// Mitsubishi GX Works2 project: Project-2_찐   PLC: Q03UD

PROGRAM AGV
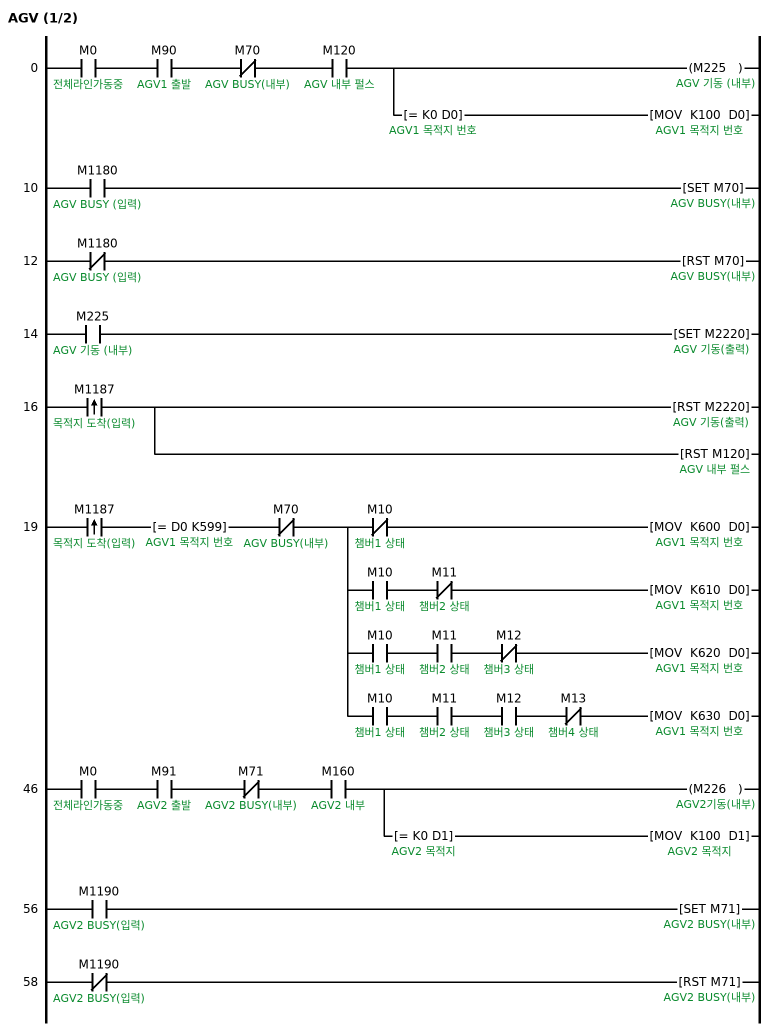
0     LD      M0  ; 전체라인가동중
      AND     M90  ; AGV1 출발
      ANI     M70  ; AGV BUSY(내부)
      AND     M120  ; AGV 내부 펄스
      OUT     M225  ; AGV 기동 (내부)
      AND=    K0 D0  ; AGV1 목적지 번호
      MOV     K100 D0
10    LD      M1180  ; AGV BUSY (입력)
      SET     M70  ; AGV BUSY(내부)
12    LDI     M1180  ; AGV BUSY (입력)
      RST     M70  ; AGV BUSY(내부)
14    LD      M225  ; AGV 기동 (내부)
      SET     M2220  ; AGV 기동(출력)
16    LDP     M1187  ; 목적지 도착(입력)
      RST     M2220  ; AGV 기동(출력)
      RST     M120  ; AGV 내부 펄스
19    LDP     M1187  ; 목적지 도착(입력)
      AND=    D0 K599  ; AGV1 목적지 번호
      ANI     M70  ; AGV BUSY(내부)
      MPS
      ANI     M10  ; 챔버1 상태
      MOV     K600 D0
      MRD
      AND     M10  ; 챔버1 상태
      ANI     M11  ; 챔버2 상태
      MOV     K610 D0
      MRD
      AND     M10  ; 챔버1 상태
      AND     M11  ; 챔버2 상태
      ANI     M12  ; 챔버3 상태
      MOV     K620 D0
      MPP
      AND     M10  ; 챔버1 상태
      AND     M11  ; 챔버2 상태
      AND     M12  ; 챔버3 상태
      ANI     M13  ; 챔버4 상태
      MOV     K630 D0
46    LD      M0  ; 전체라인가동중
      AND     M91  ; AGV2 출발
      ANI     M71  ; AGV2 BUSY(내부)
      AND     M160  ; AGV2 내부
      OUT     M226  ; AGV2기동(내부)
      AND=    K0 D1  ; AGV2 목적지
      MOV     K100 D1
56    LD      M1190  ; AGV2 BUSY(입력)
      SET     M71  ; AGV2 BUSY(내부)
58    LDI     M1190  ; AGV2 BUSY(입력)
      RST     M71  ; AGV2 BUSY(내부)
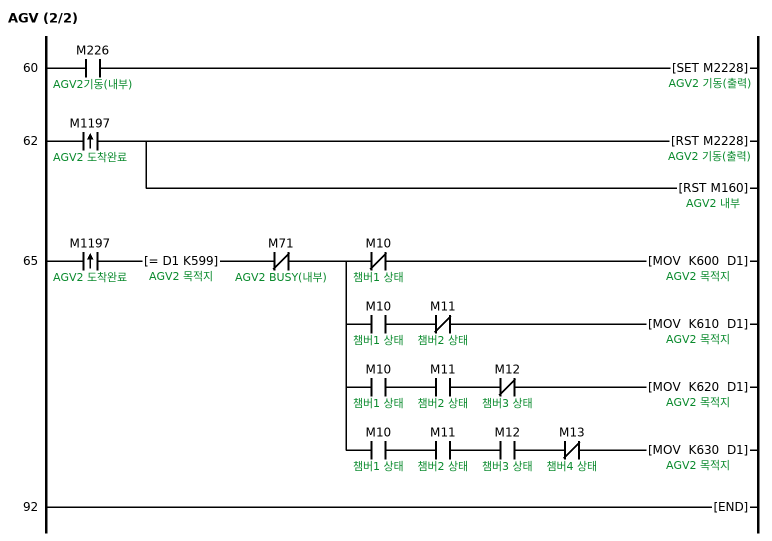
60    LD      M226  ; AGV2기동(내부)
      SET     M2228  ; AGV2 기동(출력)
62    LDP     M1197  ; AGV2 도착완료
      RST     M2228  ; AGV2 기동(출력)
      RST     M160  ; AGV2 내부
65    LDP     M1197  ; AGV2 도착완료
      AND=    D1 K599  ; AGV2 목적지
      ANI     M71  ; AGV2 BUSY(내부)
      MPS
      ANI     M10  ; 챔버1 상태
      MOV     K600 D1
      MRD
      AND     M10  ; 챔버1 상태
      ANI     M11  ; 챔버2 상태
      MOV     K610 D1
      MRD
      AND     M10  ; 챔버1 상태
      AND     M11  ; 챔버2 상태
      ANI     M12  ; 챔버3 상태
      MOV     K620 D1
      MPP
      AND     M10  ; 챔버1 상태
      AND     M11  ; 챔버2 상태
      AND     M12  ; 챔버3 상태
      ANI     M13  ; 챔버4 상태
      MOV     K630 D1
92    END
END_PROGRAM

PROGRAM Check_4
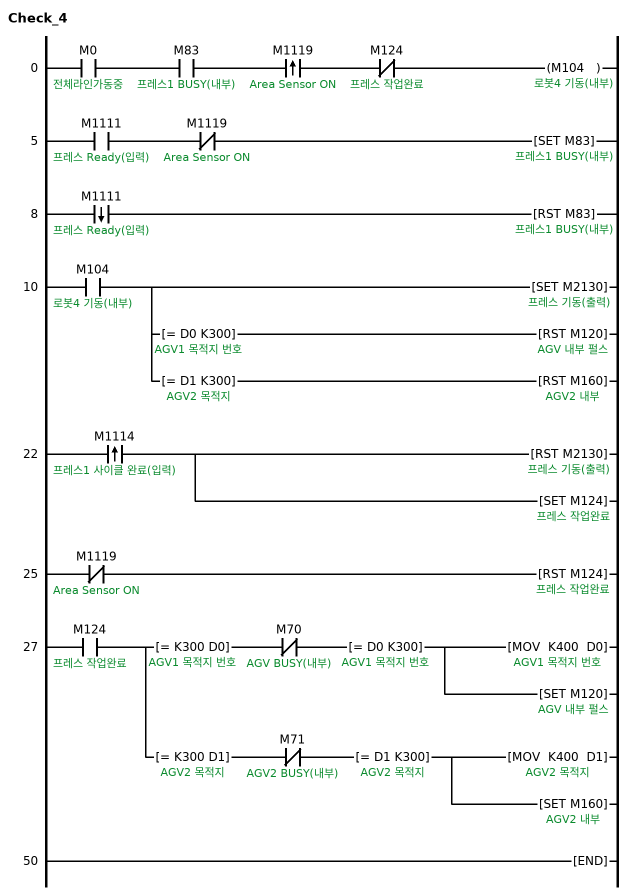
0     LD      M0  ; 전체라인가동중
      AND     M83  ; 프레스1 BUSY(내부)
      ANDP    M1119  ; Area Sensor ON
      ANI     M124  ; 프레스 작업완료
      OUT     M104  ; 로봇4 기동(내부)
5     LD      M1111  ; 프레스 Ready(입력)
      ANI     M1119  ; Area Sensor ON
      SET     M83  ; 프레스1 BUSY(내부)
8     LDF     M1111  ; 프레스 Ready(입력)
      RST     M83  ; 프레스1 BUSY(내부)
10    LD      M104  ; 로봇4 기동(내부)
      SET     M2130  ; 프레스 기동(출력)
      MPS
      AND=    D0 K300  ; AGV1 목적지 번호
      RST     M120  ; AGV 내부 펄스
      MPP
      AND=    D1 K300  ; AGV2 목적지
      RST     M160  ; AGV2 내부
22    LDP     M1114  ; 프레스1 사이클 완료(입력)
      RST     M2130  ; 프레스 기동(출력)
      SET     M124  ; 프레스 작업완료
25    LDI     M1119  ; Area Sensor ON
      RST     M124  ; 프레스 작업완료
27    LD      M124  ; 프레스 작업완료
      MPS
      AND=    K300 D0  ; AGV1 목적지 번호
      ANI     M70  ; AGV BUSY(내부)
      AND=    D0 K300  ; AGV1 목적지 번호
      MOV     K400 D0
      SET     M120  ; AGV 내부 펄스
      MPP
      AND=    K300 D1  ; AGV2 목적지
      ANI     M71  ; AGV2 BUSY(내부)
      AND=    D1 K300  ; AGV2 목적지
      MOV     K400 D1
      SET     M160  ; AGV2 내부
50    END
END_PROGRAM

PROGRAM MAIN
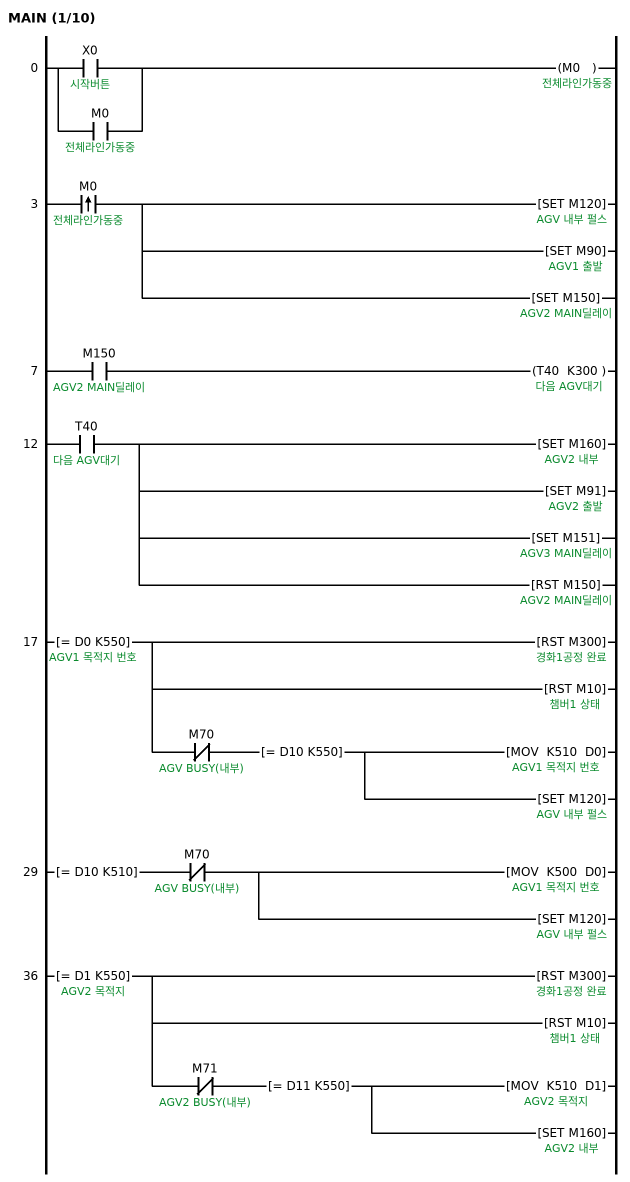
0     LD      X0  ; 시작버튼
      OR      M0  ; 전체라인가동중
      OUT     M0  ; 전체라인가동중
3     LDP     M0  ; 전체라인가동중
      SET     M120  ; AGV 내부 펄스
      SET     M90  ; AGV1 출발
      SET     M150  ; AGV2 MAIN딜레이
7     LD      M150  ; AGV2 MAIN딜레이
      OUT     T40 K300  ; 다음 AGV대기
12    LD      T40  ; 다음 AGV대기
      SET     M160  ; AGV2 내부
      SET     M91  ; AGV2 출발
      SET     M151  ; AGV3 MAIN딜레이
      RST     M150  ; AGV2 MAIN딜레이
17    LD=     D0 K550  ; AGV1 목적지 번호
      RST     M300  ; 경화1공정 완료
      RST     M10  ; 챔버1 상태
      ANI     M70  ; AGV BUSY(내부)
      AND=    D10 K550
      MOV     K510 D0
      SET     M120  ; AGV 내부 펄스
29    LD=     D10 K510
      ANI     M70  ; AGV BUSY(내부)
      MOV     K500 D0
      SET     M120  ; AGV 내부 펄스
36    LD=     D1 K550  ; AGV2 목적지
      RST     M300  ; 경화1공정 완료
      RST     M10  ; 챔버1 상태
      ANI     M71  ; AGV2 BUSY(내부)
      AND=    D11 K550
      MOV     K510 D1
      SET     M160  ; AGV2 내부
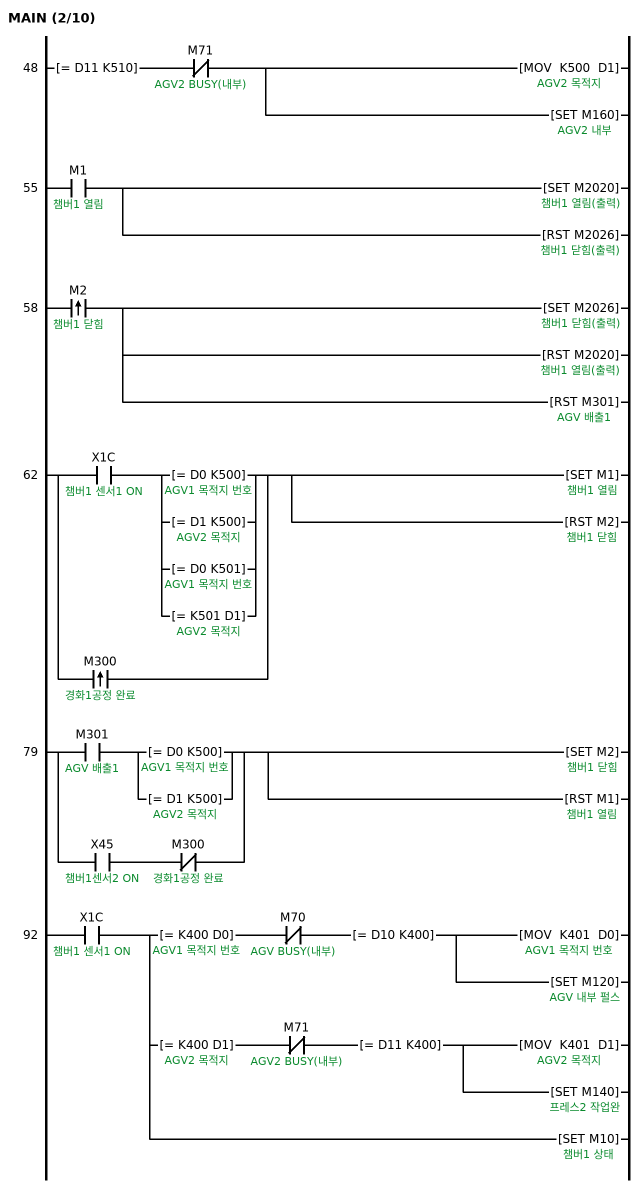
48    LD=     D11 K510
      ANI     M71  ; AGV2 BUSY(내부)
      MOV     K500 D1
      SET     M160  ; AGV2 내부
55    LD      M1  ; 챔버1 열림
      SET     M2020  ; 챔버1 열림(출력)
      RST     M2026  ; 챔버1 닫힘(출력)
58    LDP     M2  ; 챔버1 닫힘
      SET     M2026  ; 챔버1 닫힘(출력)
      RST     M2020  ; 챔버1 열림(출력)
      RST     M301  ; AGV 배출1
62    LD      X1C  ; 챔버1 센서1 ON
      LD=     D0 K500  ; AGV1 목적지 번호
      OR=     D1 K500  ; AGV2 목적지
      OR=     D0 K501  ; AGV1 목적지 번호
      OR=     K501 D1  ; AGV2 목적지
      ANB
      ORP     M300  ; 경화1공정 완료
      SET     M1  ; 챔버1 열림
      RST     M2  ; 챔버1 닫힘
79    LD      M301  ; AGV 배출1
      LD=     D0 K500  ; AGV1 목적지 번호
      OR=     D1 K500  ; AGV2 목적지
      ANB
      LD      X45  ; 챔버1센서2 ON
      ANI     M300  ; 경화1공정 완료
      ORB
      SET     M2  ; 챔버1 닫힘
      RST     M1  ; 챔버1 열림
92    LD      X1C  ; 챔버1 센서1 ON
      MPS
      AND=    K400 D0  ; AGV1 목적지 번호
      ANI     M70  ; AGV BUSY(내부)
      AND=    D10 K400
      MOV     K401 D0
      SET     M120  ; AGV 내부 펄스
      MRD
      AND=    K400 D1  ; AGV2 목적지
      ANI     M71  ; AGV2 BUSY(내부)
      AND=    D11 K400
      MOV     K401 D1
      SET     M140  ; 프레스2 작업완
      MPP
      SET     M10  ; 챔버1 상태
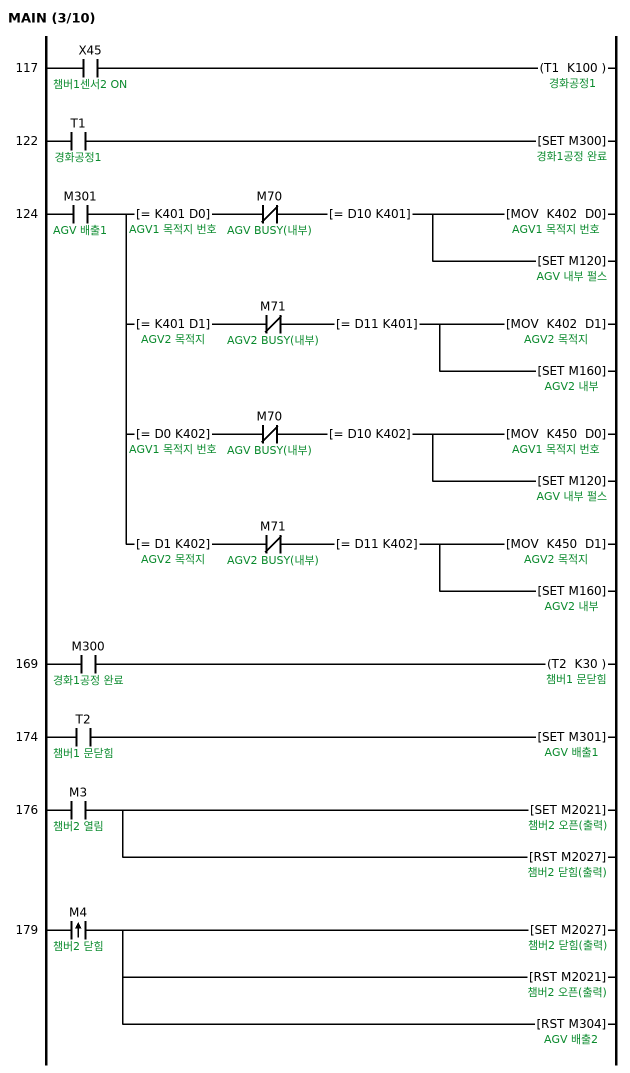
117   LD      X45  ; 챔버1센서2 ON
      OUT     T1 K100  ; 경화공정1
122   LD      T1  ; 경화공정1
      SET     M300  ; 경화1공정 완료
124   LD      M301  ; AGV 배출1
      MPS
      AND=    K401 D0  ; AGV1 목적지 번호
      ANI     M70  ; AGV BUSY(내부)
      AND=    D10 K401
      MOV     K402 D0
      SET     M120  ; AGV 내부 펄스
      MRD
      AND=    K401 D1  ; AGV2 목적지
      ANI     M71  ; AGV2 BUSY(내부)
      AND=    D11 K401
      MOV     K402 D1
      SET     M160  ; AGV2 내부
      MRD
      AND=    D0 K402  ; AGV1 목적지 번호
      ANI     M70  ; AGV BUSY(내부)
      AND=    D10 K402
      MOV     K450 D0
      SET     M120  ; AGV 내부 펄스
      MPP
      AND=    D1 K402  ; AGV2 목적지
      ANI     M71  ; AGV2 BUSY(내부)
      AND=    D11 K402
      MOV     K450 D1
      SET     M160  ; AGV2 내부
169   LD      M300  ; 경화1공정 완료
      OUT     T2 K30  ; 챔버1 문닫힘
174   LD      T2  ; 챔버1 문닫힘
      SET     M301  ; AGV 배출1
176   LD      M3  ; 챔버2 열림
      SET     M2021  ; 챔버2 오픈(출력)
      RST     M2027  ; 챔버2 닫힘(출력)
179   LDP     M4  ; 챔버2 닫힘
      SET     M2027  ; 챔버2 닫힘(출력)
      RST     M2021  ; 챔버2 오픈(출력)
      RST     M304  ; AGV 배출2
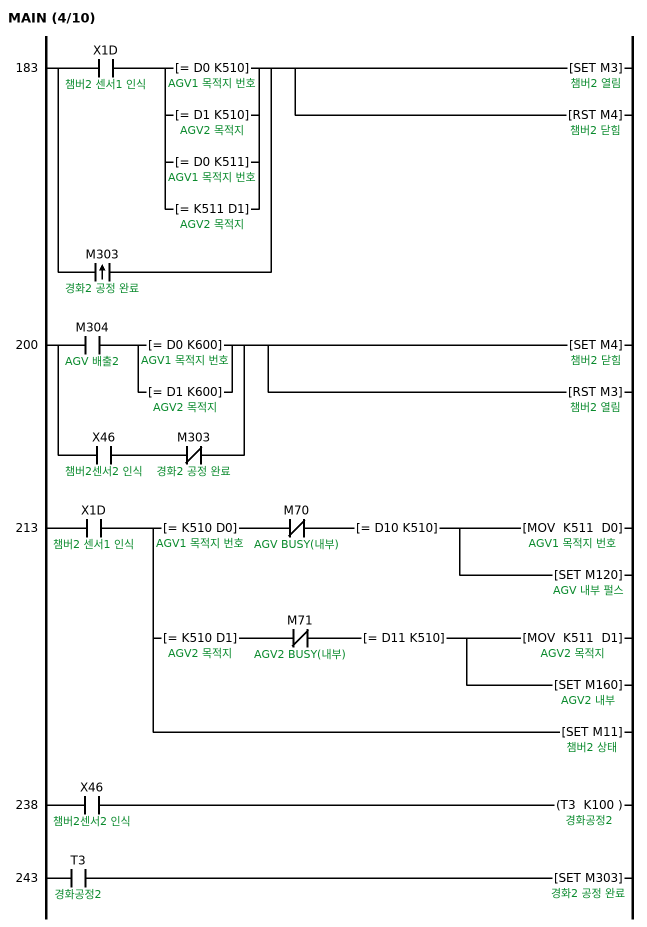
183   LD      X1D  ; 챔버2 센서1 인식
      LD=     D0 K510  ; AGV1 목적지 번호
      OR=     D1 K510  ; AGV2 목적지
      OR=     D0 K511  ; AGV1 목적지 번호
      OR=     K511 D1  ; AGV2 목적지
      ANB
      ORP     M303  ; 경화2 공정 완료
      SET     M3  ; 챔버2 열림
      RST     M4  ; 챔버2 닫힘
200   LD      M304  ; AGV 배출2
      LD=     D0 K600  ; AGV1 목적지 번호
      OR=     D1 K600  ; AGV2 목적지
      ANB
      LD      X46  ; 챔버2센서2 인식
      ANI     M303  ; 경화2 공정 완료
      ORB
      SET     M4  ; 챔버2 닫힘
      RST     M3  ; 챔버2 열림
213   LD      X1D  ; 챔버2 센서1 인식
      MPS
      AND=    K510 D0  ; AGV1 목적지 번호
      ANI     M70  ; AGV BUSY(내부)
      AND=    D10 K510
      MOV     K511 D0
      SET     M120  ; AGV 내부 펄스
      MRD
      AND=    K510 D1  ; AGV2 목적지
      ANI     M71  ; AGV2 BUSY(내부)
      AND=    D11 K510
      MOV     K511 D1
      SET     M160  ; AGV2 내부
      MPP
      SET     M11  ; 챔버2 상태
238   LD      X46  ; 챔버2센서2 인식
      OUT     T3 K100  ; 경화공정2
243   LD      T3  ; 경화공정2
      SET     M303  ; 경화2 공정 완료
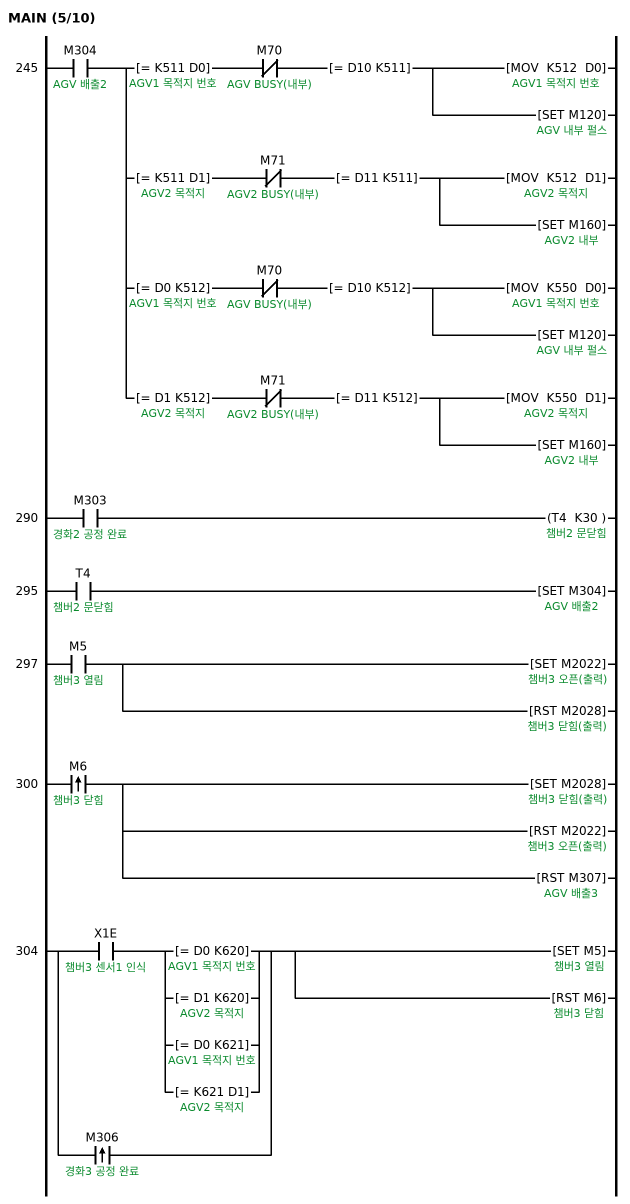
245   LD      M304  ; AGV 배출2
      MPS
      AND=    K511 D0  ; AGV1 목적지 번호
      ANI     M70  ; AGV BUSY(내부)
      AND=    D10 K511
      MOV     K512 D0
      SET     M120  ; AGV 내부 펄스
      MRD
      AND=    K511 D1  ; AGV2 목적지
      ANI     M71  ; AGV2 BUSY(내부)
      AND=    D11 K511
      MOV     K512 D1
      SET     M160  ; AGV2 내부
      MRD
      AND=    D0 K512  ; AGV1 목적지 번호
      ANI     M70  ; AGV BUSY(내부)
      AND=    D10 K512
      MOV     K550 D0
      SET     M120  ; AGV 내부 펄스
      MPP
      AND=    D1 K512  ; AGV2 목적지
      ANI     M71  ; AGV2 BUSY(내부)
      AND=    D11 K512
      MOV     K550 D1
      SET     M160  ; AGV2 내부
290   LD      M303  ; 경화2 공정 완료
      OUT     T4 K30  ; 챔버2 문닫힘
295   LD      T4  ; 챔버2 문닫힘
      SET     M304  ; AGV 배출2
297   LD      M5  ; 챔버3 열림
      SET     M2022  ; 챔버3 오픈(출력)
      RST     M2028  ; 챔버3 닫힘(출력)
300   LDP     M6  ; 챔버3 닫힘
      SET     M2028  ; 챔버3 닫힘(출력)
      RST     M2022  ; 챔버3 오픈(출력)
      RST     M307  ; AGV 배출3
304   LD      X1E  ; 챔버3 센서1 인식
      LD=     D0 K620  ; AGV1 목적지 번호
      OR=     D1 K620  ; AGV2 목적지
      OR=     D0 K621  ; AGV1 목적지 번호
      OR=     K621 D1  ; AGV2 목적지
      ANB
      ORP     M306  ; 경화3 공정 완료
      SET     M5  ; 챔버3 열림
      RST     M6  ; 챔버3 닫힘
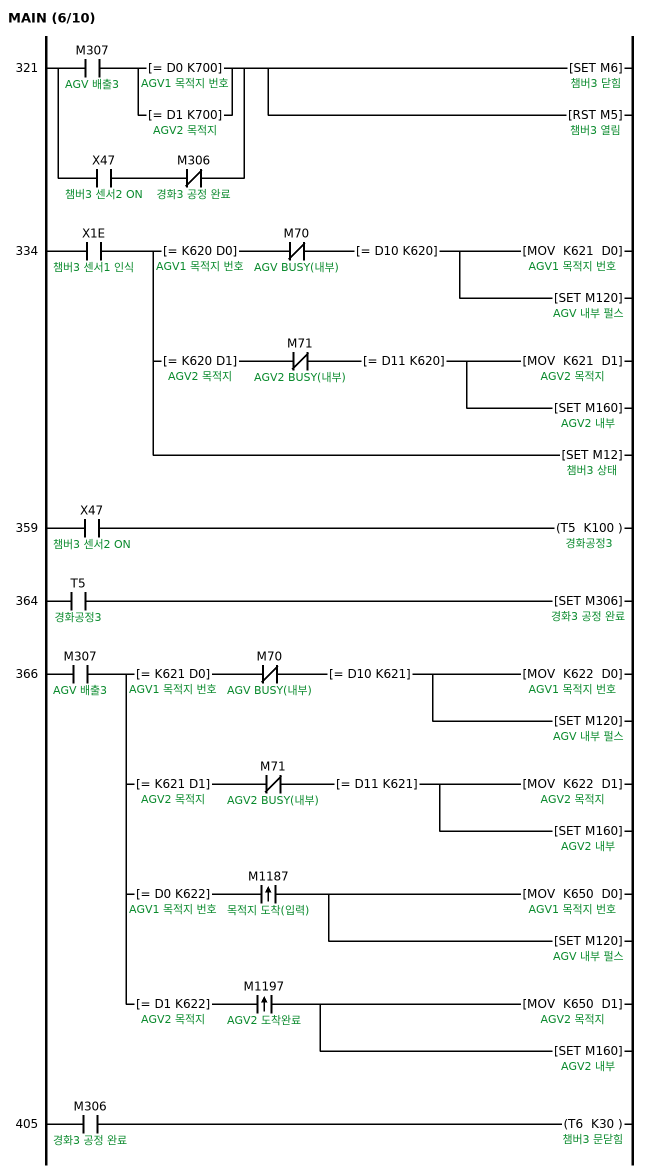
321   LD      M307  ; AGV 배출3
      LD=     D0 K700  ; AGV1 목적지 번호
      OR=     D1 K700  ; AGV2 목적지
      ANB
      LD      X47  ; 챔버3 센서2 ON
      ANI     M306  ; 경화3 공정 완료
      ORB
      SET     M6  ; 챔버3 닫힘
      RST     M5  ; 챔버3 열림
334   LD      X1E  ; 챔버3 센서1 인식
      MPS
      AND=    K620 D0  ; AGV1 목적지 번호
      ANI     M70  ; AGV BUSY(내부)
      AND=    D10 K620
      MOV     K621 D0
      SET     M120  ; AGV 내부 펄스
      MRD
      AND=    K620 D1  ; AGV2 목적지
      ANI     M71  ; AGV2 BUSY(내부)
      AND=    D11 K620
      MOV     K621 D1
      SET     M160  ; AGV2 내부
      MPP
      SET     M12  ; 챔버3 상태
359   LD      X47  ; 챔버3 센서2 ON
      OUT     T5 K100  ; 경화공정3
364   LD      T5  ; 경화공정3
      SET     M306  ; 경화3 공정 완료
366   LD      M307  ; AGV 배출3
      MPS
      AND=    K621 D0  ; AGV1 목적지 번호
      ANI     M70  ; AGV BUSY(내부)
      AND=    D10 K621
      MOV     K622 D0
      SET     M120  ; AGV 내부 펄스
      MRD
      AND=    K621 D1  ; AGV2 목적지
      ANI     M71  ; AGV2 BUSY(내부)
      AND=    D11 K621
      MOV     K622 D1
      SET     M160  ; AGV2 내부
      MRD
      AND=    D0 K622  ; AGV1 목적지 번호
      ANDP    M1187  ; 목적지 도착(입력)
      MOV     K650 D0
      SET     M120  ; AGV 내부 펄스
      MPP
      AND=    D1 K622  ; AGV2 목적지
      ANDP    M1197  ; AGV2 도착완료
      MOV     K650 D1
      SET     M160  ; AGV2 내부
405   LD      M306  ; 경화3 공정 완료
      OUT     T6 K30  ; 챔버3 문닫힘
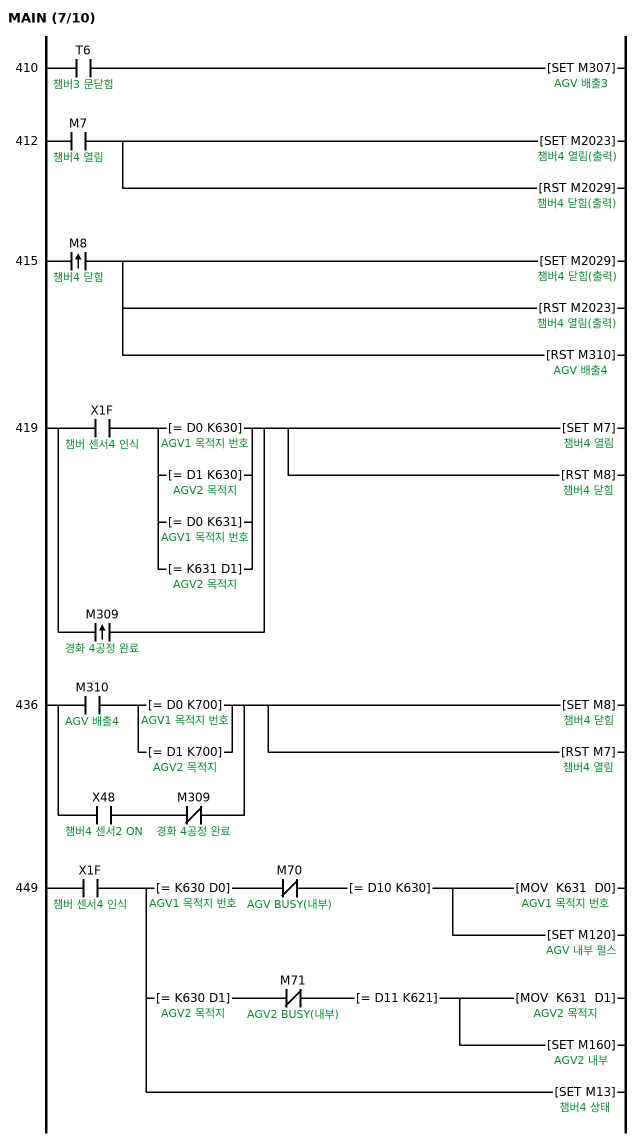
410   LD      T6  ; 챔버3 문닫힘
      SET     M307  ; AGV 배출3
412   LD      M7  ; 챔버4 열림
      SET     M2023  ; 챔버4 열림(출력)
      RST     M2029  ; 챔버4 닫힘(출력)
415   LDP     M8  ; 챔버4 닫힘
      SET     M2029  ; 챔버4 닫힘(출력)
      RST     M2023  ; 챔버4 열림(출력)
      RST     M310  ; AGV 배출4
419   LD      X1F  ; 챔버 센서4 인식
      LD=     D0 K630  ; AGV1 목적지 번호
      OR=     D1 K630  ; AGV2 목적지
      OR=     D0 K631  ; AGV1 목적지 번호
      OR=     K631 D1  ; AGV2 목적지
      ANB
      ORP     M309  ; 경화 4공정 완료
      SET     M7  ; 챔버4 열림
      RST     M8  ; 챔버4 닫힘
436   LD      M310  ; AGV 배출4
      LD=     D0 K700  ; AGV1 목적지 번호
      OR=     D1 K700  ; AGV2 목적지
      ANB
      LD      X48  ; 챔버4 센서2 ON
      ANI     M309  ; 경화 4공정 완료
      ORB
      SET     M8  ; 챔버4 닫힘
      RST     M7  ; 챔버4 열림
449   LD      X1F  ; 챔버 센서4 인식
      MPS
      AND=    K630 D0  ; AGV1 목적지 번호
      ANI     M70  ; AGV BUSY(내부)
      AND=    D10 K630
      MOV     K631 D0
      SET     M120  ; AGV 내부 펄스
      MRD
      AND=    K630 D1  ; AGV2 목적지
      ANI     M71  ; AGV2 BUSY(내부)
      AND=    D11 K621
      MOV     K631 D1
      SET     M160  ; AGV2 내부
      MPP
      SET     M13  ; 챔버4 상태
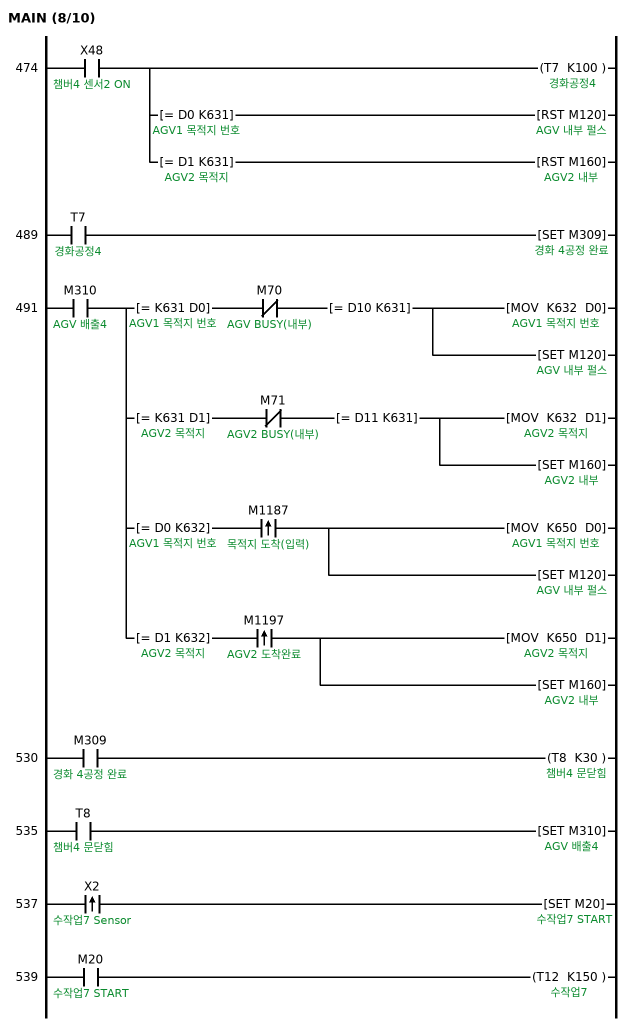
474   LD      X48  ; 챔버4 센서2 ON
      OUT     T7 K100  ; 경화공정4
      MPS
      AND=    D0 K631  ; AGV1 목적지 번호
      RST     M120  ; AGV 내부 펄스
      MPP
      AND=    D1 K631  ; AGV2 목적지
      RST     M160  ; AGV2 내부
489   LD      T7  ; 경화공정4
      SET     M309  ; 경화 4공정 완료
491   LD      M310  ; AGV 배출4
      MPS
      AND=    K631 D0  ; AGV1 목적지 번호
      ANI     M70  ; AGV BUSY(내부)
      AND=    D10 K631
      MOV     K632 D0
      SET     M120  ; AGV 내부 펄스
      MRD
      AND=    K631 D1  ; AGV2 목적지
      ANI     M71  ; AGV2 BUSY(내부)
      AND=    D11 K631
      MOV     K632 D1
      SET     M160  ; AGV2 내부
      MRD
      AND=    D0 K632  ; AGV1 목적지 번호
      ANDP    M1187  ; 목적지 도착(입력)
      MOV     K650 D0
      SET     M120  ; AGV 내부 펄스
      MPP
      AND=    D1 K632  ; AGV2 목적지
      ANDP    M1197  ; AGV2 도착완료
      MOV     K650 D1
      SET     M160  ; AGV2 내부
530   LD      M309  ; 경화 4공정 완료
      OUT     T8 K30  ; 챔버4 문닫힘
535   LD      T8  ; 챔버4 문닫힘
      SET     M310  ; AGV 배출4
537   LDP     X2  ; 수작업7 Sensor
      SET     M20  ; 수작업7 START
539   LD      M20  ; 수작업7 START
      OUT     T12 K150  ; 수작업7
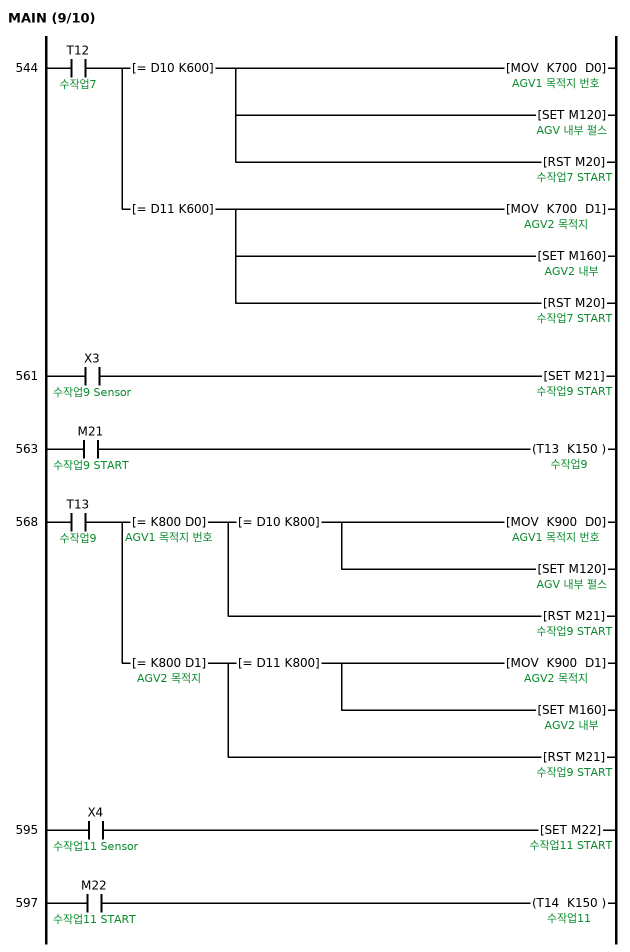
544   LD      T12  ; 수작업7
      MPS
      AND=    D10 K600
      MOV     K700 D0
      SET     M120  ; AGV 내부 펄스
      RST     M20  ; 수작업7 START
      MPP
      AND=    D11 K600
      MOV     K700 D1
      SET     M160  ; AGV2 내부
      RST     M20  ; 수작업7 START
561   LD      X3  ; 수작업9 Sensor
      SET     M21  ; 수작업9 START
563   LD      M21  ; 수작업9 START
      OUT     T13 K150  ; 수작업9
568   LD      T13  ; 수작업9
      MPS
      AND=    K800 D0  ; AGV1 목적지 번호
      MPS
      AND=    D10 K800
      MOV     K900 D0
      SET     M120  ; AGV 내부 펄스
      MPP
      RST     M21  ; 수작업9 START
      MPP
      AND=    K800 D1  ; AGV2 목적지
      MPS
      AND=    D11 K800
      MOV     K900 D1
      SET     M160  ; AGV2 내부
      MPP
      RST     M21  ; 수작업9 START
595   LD      X4  ; 수작업11 Sensor
      SET     M22  ; 수작업11 START
597   LD      M22  ; 수작업11 START
      OUT     T14 K150  ; 수작업11
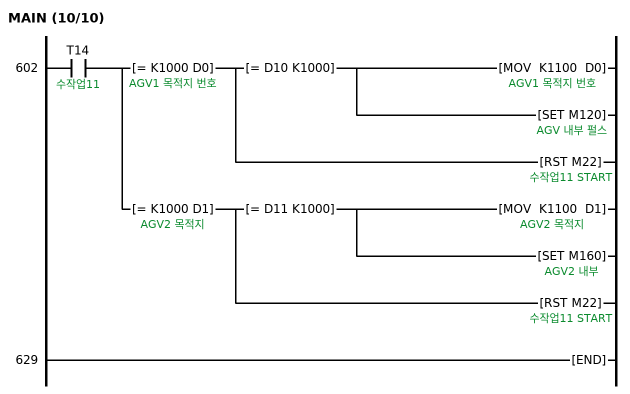
602   LD      T14  ; 수작업11
      MPS
      AND=    K1000 D0  ; AGV1 목적지 번호
      MPS
      AND=    D10 K1000
      MOV     K1100 D0
      SET     M120  ; AGV 내부 펄스
      MPP
      RST     M22  ; 수작업11 START
      MPP
      AND=    K1000 D1  ; AGV2 목적지
      MPS
      AND=    D11 K1000
      MOV     K1100 D1
      SET     M160  ; AGV2 내부
      MPP
      RST     M22  ; 수작업11 START
629   END
END_PROGRAM

PROGRAM Press_10
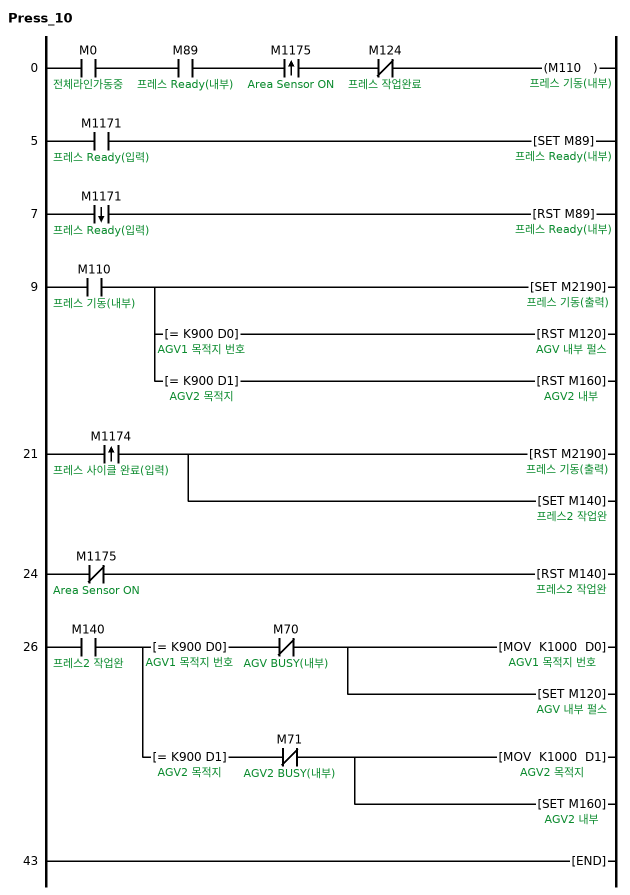
0     LD      M0  ; 전체라인가동중
      AND     M89  ; 프레스 Ready(내부)
      ANDP    M1175  ; Area Sensor ON
      ANI     M124  ; 프레스 작업완료
      OUT     M110  ; 프레스 기동(내부)
5     LD      M1171  ; 프레스 Ready(입력)
      SET     M89  ; 프레스 Ready(내부)
7     LDF     M1171  ; 프레스 Ready(입력)
      RST     M89  ; 프레스 Ready(내부)
9     LD      M110  ; 프레스 기동(내부)
      SET     M2190  ; 프레스 기동(출력)
      MPS
      AND=    K900 D0  ; AGV1 목적지 번호
      RST     M120  ; AGV 내부 펄스
      MPP
      AND=    K900 D1  ; AGV2 목적지
      RST     M160  ; AGV2 내부
21    LDP     M1174  ; 프레스 사이클 완료(입력)
      RST     M2190  ; 프레스 기동(출력)
      SET     M140  ; 프레스2 작업완
24    LDI     M1175  ; Area Sensor ON
      RST     M140  ; 프레스2 작업완
26    LD      M140  ; 프레스2 작업완
      MPS
      AND=    K900 D0  ; AGV1 목적지 번호
      ANI     M70  ; AGV BUSY(내부)
      MOV     K1000 D0
      SET     M120  ; AGV 내부 펄스
      MPP
      AND=    K900 D1  ; AGV2 목적지
      ANI     M71  ; AGV2 BUSY(내부)
      MOV     K1000 D1
      SET     M160  ; AGV2 내부
43    END
END_PROGRAM

PROGRAM Rob1_1
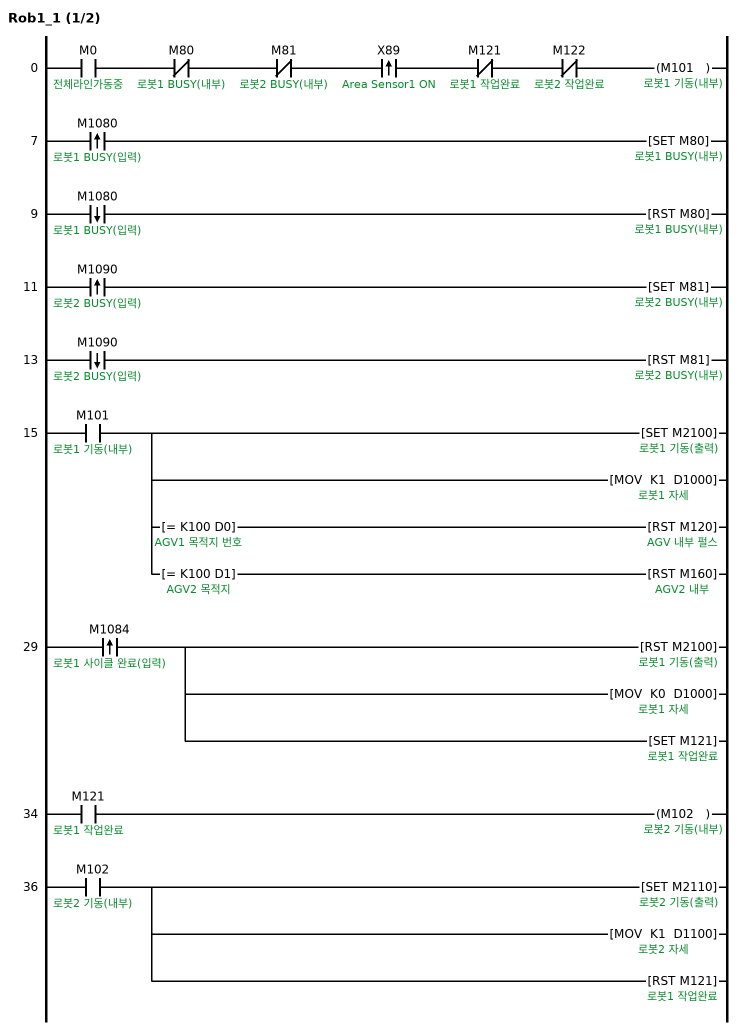
0     LD      M0  ; 전체라인가동중
      ANI     M80  ; 로봇1 BUSY(내부)
      ANI     M81  ; 로봇2 BUSY(내부)
      ANDP    X89  ; Area Sensor1 ON
      ANI     M121  ; 로봇1 작업완료
      ANI     M122  ; 로봇2 작업완료
      OUT     M101  ; 로봇1 기동(내부)
7     LDP     M1080  ; 로봇1 BUSY(입력)
      SET     M80  ; 로봇1 BUSY(내부)
9     LDF     M1080  ; 로봇1 BUSY(입력)
      RST     M80  ; 로봇1 BUSY(내부)
11    LDP     M1090  ; 로봇2 BUSY(입력)
      SET     M81  ; 로봇2 BUSY(내부)
13    LDF     M1090  ; 로봇2 BUSY(입력)
      RST     M81  ; 로봇2 BUSY(내부)
15    LD      M101  ; 로봇1 기동(내부)
      SET     M2100  ; 로봇1 기동(출력)
      MOV     K1 D1000  ; 로봇1 자세
      MPS
      AND=    K100 D0  ; AGV1 목적지 번호
      RST     M120  ; AGV 내부 펄스
      MPP
      AND=    K100 D1  ; AGV2 목적지
      RST     M160  ; AGV2 내부
29    LDP     M1084  ; 로봇1 사이클 완료(입력)
      RST     M2100  ; 로봇1 기동(출력)
      MOV     K0 D1000
      SET     M121  ; 로봇1 작업완료
34    LD      M121  ; 로봇1 작업완료
      OUT     M102  ; 로봇2 기동(내부)
36    LD      M102  ; 로봇2 기동(내부)
      SET     M2110  ; 로봇2 기동(출력)
      MOV     K1 D1100  ; 로봇2 자세
      RST     M121  ; 로봇1 작업완료
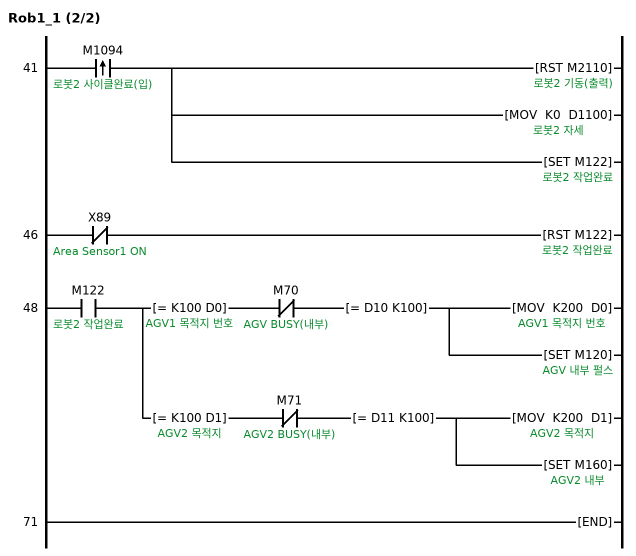
41    LDP     M1094  ; 로봇2 사이클완료(입)
      RST     M2110  ; 로봇2 기동(출력)
      MOV     K0 D1100
      SET     M122  ; 로봇2 작업완료
46    LDI     X89  ; Area Sensor1 ON
      RST     M122  ; 로봇2 작업완료
48    LD      M122  ; 로봇2 작업완료
      MPS
      AND=    K100 D0  ; AGV1 목적지 번호
      ANI     M70  ; AGV BUSY(내부)
      AND=    D10 K100
      MOV     K200 D0
      SET     M120  ; AGV 내부 펄스
      MPP
      AND=    K100 D1  ; AGV2 목적지
      ANI     M71  ; AGV2 BUSY(내부)
      AND=    D11 K100
      MOV     K200 D1
      SET     M160  ; AGV2 내부
71    END
END_PROGRAM

PROGRAM Rob3_3
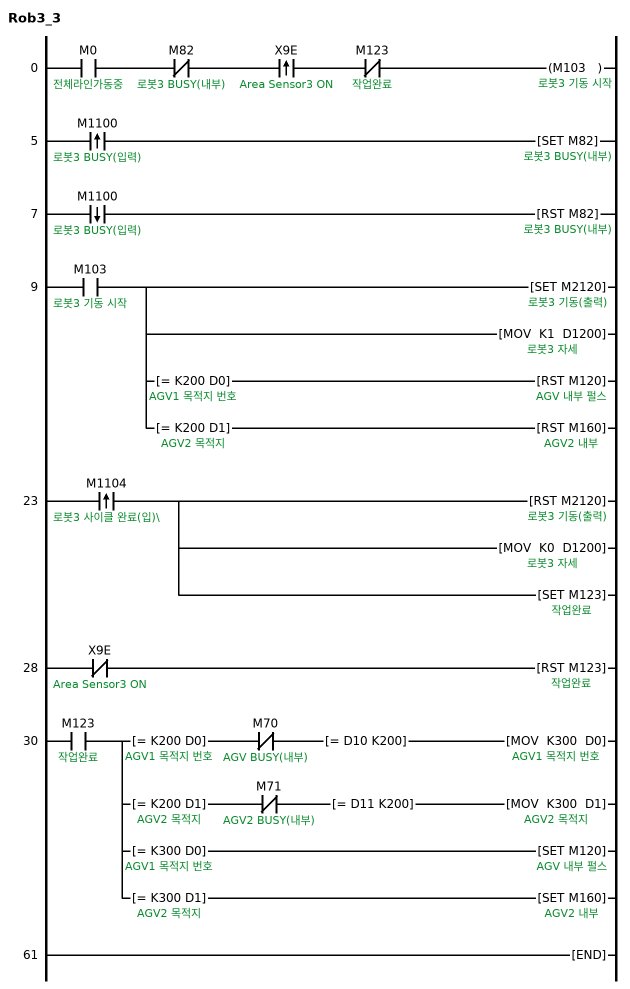
0     LD      M0  ; 전체라인가동중
      ANI     M82  ; 로봇3 BUSY(내부)
      ANDP    X9E  ; Area Sensor3 ON
      ANI     M123  ; 작업완료
      OUT     M103  ; 로봇3 기동 시작
5     LDP     M1100  ; 로봇3 BUSY(입력)
      SET     M82  ; 로봇3 BUSY(내부)
7     LDF     M1100  ; 로봇3 BUSY(입력)
      RST     M82  ; 로봇3 BUSY(내부)
9     LD      M103  ; 로봇3 기동 시작
      SET     M2120  ; 로봇3 기동(출력)
      MOV     K1 D1200  ; 로봇3 자세
      MPS
      AND=    K200 D0  ; AGV1 목적지 번호
      RST     M120  ; AGV 내부 펄스
      MPP
      AND=    K200 D1  ; AGV2 목적지
      RST     M160  ; AGV2 내부
23    LDP     M1104  ; 로봇3 사이클 완료(입)\
      RST     M2120  ; 로봇3 기동(출력)
      MOV     K0 D1200
      SET     M123  ; 작업완료
28    LDI     X9E  ; Area Sensor3 ON
      RST     M123  ; 작업완료
30    LD      M123  ; 작업완료
      MPS
      AND=    K200 D0  ; AGV1 목적지 번호
      ANI     M70  ; AGV BUSY(내부)
      AND=    D10 K200
      MOV     K300 D0
      MRD
      AND=    K200 D1  ; AGV2 목적지
      ANI     M71  ; AGV2 BUSY(내부)
      AND=    D11 K200
      MOV     K300 D1
      MRD
      AND=    K300 D0  ; AGV1 목적지 번호
      SET     M120  ; AGV 내부 펄스
      MPP
      AND=    K300 D1  ; AGV2 목적지
      SET     M160  ; AGV2 내부
61    END
END_PROGRAM

PROGRAM Rob5_5
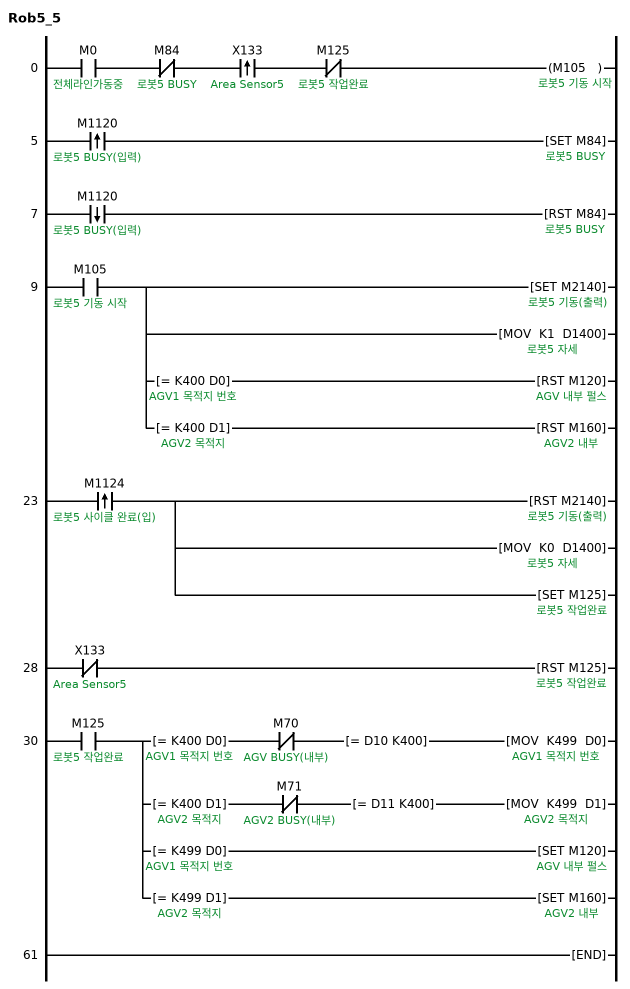
0     LD      M0  ; 전체라인가동중
      ANI     M84  ; 로봇5 BUSY
      ANDP    X133  ; Area Sensor5
      ANI     M125  ; 로봇5 작업완료
      OUT     M105  ; 로봇5 기동 시작
5     LDP     M1120  ; 로봇5 BUSY(입력)
      SET     M84  ; 로봇5 BUSY
7     LDF     M1120  ; 로봇5 BUSY(입력)
      RST     M84  ; 로봇5 BUSY
9     LD      M105  ; 로봇5 기동 시작
      SET     M2140  ; 로봇5 기동(출력)
      MOV     K1 D1400  ; 로봇5 자세
      MPS
      AND=    K400 D0  ; AGV1 목적지 번호
      RST     M120  ; AGV 내부 펄스
      MPP
      AND=    K400 D1  ; AGV2 목적지
      RST     M160  ; AGV2 내부
23    LDP     M1124  ; 로봇5 사이클 완료(입)
      RST     M2140  ; 로봇5 기동(출력)
      MOV     K0 D1400
      SET     M125  ; 로봇5 작업완료
28    LDI     X133  ; Area Sensor5
      RST     M125  ; 로봇5 작업완료
30    LD      M125  ; 로봇5 작업완료
      MPS
      AND=    K400 D0  ; AGV1 목적지 번호
      ANI     M70  ; AGV BUSY(내부)
      AND=    D10 K400
      MOV     K499 D0
      MRD
      AND=    K400 D1  ; AGV2 목적지
      ANI     M71  ; AGV2 BUSY(내부)
      AND=    D11 K400
      MOV     K499 D1
      MRD
      AND=    K499 D0  ; AGV1 목적지 번호
      SET     M120  ; AGV 내부 펄스
      MPP
      AND=    K499 D1  ; AGV2 목적지
      SET     M160  ; AGV2 내부
61    END
END_PROGRAM

PROGRAM Rob6_8
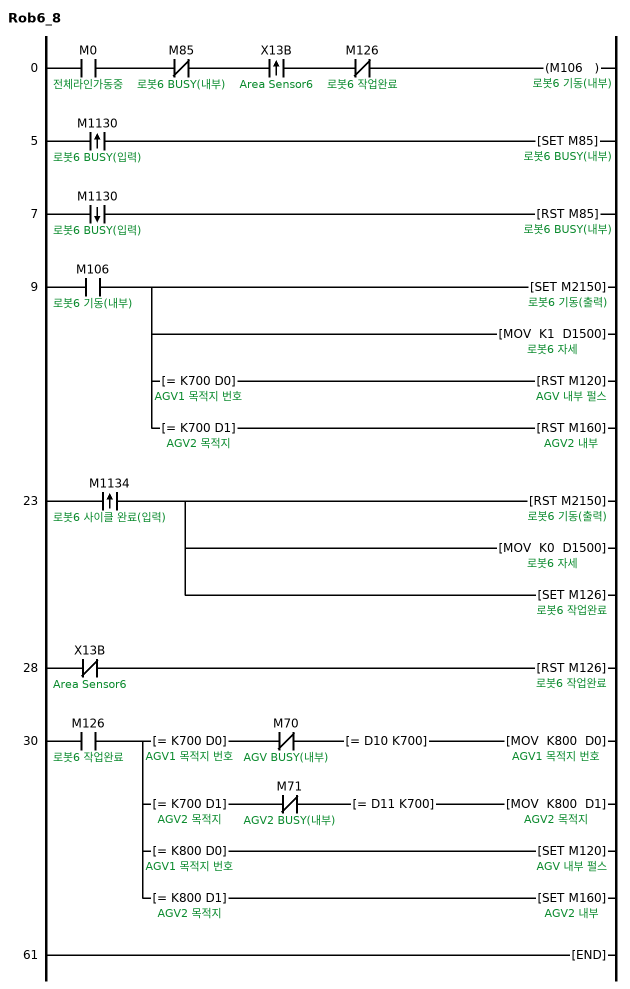
0     LD      M0  ; 전체라인가동중
      ANI     M85  ; 로봇6 BUSY(내부)
      ANDP    X13B  ; Area Sensor6
      ANI     M126  ; 로봇6 작업완료
      OUT     M106  ; 로봇6 기동(내부)
5     LDP     M1130  ; 로봇6 BUSY(입력)
      SET     M85  ; 로봇6 BUSY(내부)
7     LDF     M1130  ; 로봇6 BUSY(입력)
      RST     M85  ; 로봇6 BUSY(내부)
9     LD      M106  ; 로봇6 기동(내부)
      SET     M2150  ; 로봇6 기동(출력)
      MOV     K1 D1500  ; 로봇6 자세
      MPS
      AND=    K700 D0  ; AGV1 목적지 번호
      RST     M120  ; AGV 내부 펄스
      MPP
      AND=    K700 D1  ; AGV2 목적지
      RST     M160  ; AGV2 내부
23    LDP     M1134  ; 로봇6 사이클 완료(입력)
      RST     M2150  ; 로봇6 기동(출력)
      MOV     K0 D1500
      SET     M126  ; 로봇6 작업완료
28    LDI     X13B  ; Area Sensor6
      RST     M126  ; 로봇6 작업완료
30    LD      M126  ; 로봇6 작업완료
      MPS
      AND=    K700 D0  ; AGV1 목적지 번호
      ANI     M70  ; AGV BUSY(내부)
      AND=    D10 K700
      MOV     K800 D0
      MRD
      AND=    K700 D1  ; AGV2 목적지
      ANI     M71  ; AGV2 BUSY(내부)
      AND=    D11 K700
      MOV     K800 D1
      MRD
      AND=    K800 D0  ; AGV1 목적지 번호
      SET     M120  ; AGV 내부 펄스
      MPP
      AND=    K800 D1  ; AGV2 목적지
      SET     M160  ; AGV2 내부
61    END
END_PROGRAM

PROGRAM Rob9_13
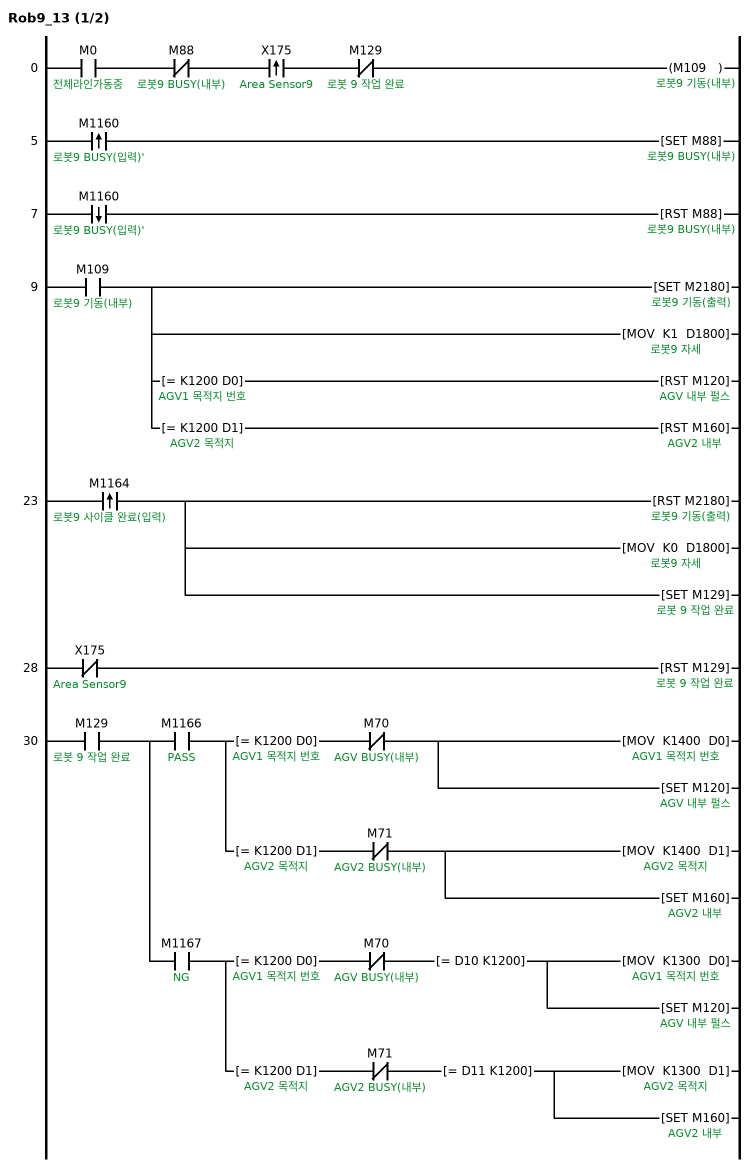
0     LD      M0  ; 전체라인가동중
      ANI     M88  ; 로봇9 BUSY(내부)
      ANDP    X175  ; Area Sensor9
      ANI     M129  ; 로봇 9 작업 완료
      OUT     M109  ; 로봇9 기동(내부)
5     LDP     M1160  ; 로봇9 BUSY(입력)'
      SET     M88  ; 로봇9 BUSY(내부)
7     LDF     M1160  ; 로봇9 BUSY(입력)'
      RST     M88  ; 로봇9 BUSY(내부)
9     LD      M109  ; 로봇9 기동(내부)
      SET     M2180  ; 로봇9 기동(출력)
      MOV     K1 D1800  ; 로봇9 자세
      MPS
      AND=    K1200 D0  ; AGV1 목적지 번호
      RST     M120  ; AGV 내부 펄스
      MPP
      AND=    K1200 D1  ; AGV2 목적지
      RST     M160  ; AGV2 내부
23    LDP     M1164  ; 로봇9 사이클 완료(입력)
      RST     M2180  ; 로봇9 기동(출력)
      MOV     K0 D1800
      SET     M129  ; 로봇 9 작업 완료
28    LDI     X175  ; Area Sensor9
      RST     M129  ; 로봇 9 작업 완료
30    LD      M129  ; 로봇 9 작업 완료
      MPS
      AND     M1166  ; PASS
      MPS
      AND=    K1200 D0  ; AGV1 목적지 번호
      ANI     M70  ; AGV BUSY(내부)
      MOV     K1400 D0
      SET     M120  ; AGV 내부 펄스
      MPP
      AND=    K1200 D1  ; AGV2 목적지
      ANI     M71  ; AGV2 BUSY(내부)
      MOV     K1400 D1
      SET     M160  ; AGV2 내부
      MPP
      AND     M1167  ; NG
      MPS
      AND=    K1200 D0  ; AGV1 목적지 번호
      ANI     M70  ; AGV BUSY(내부)
      AND=    D10 K1200
      MOV     K1300 D0
      SET     M120  ; AGV 내부 펄스
      MPP
      AND=    K1200 D1  ; AGV2 목적지
      ANI     M71  ; AGV2 BUSY(내부)
      AND=    D11 K1200
      MOV     K1300 D1
      SET     M160  ; AGV2 내부
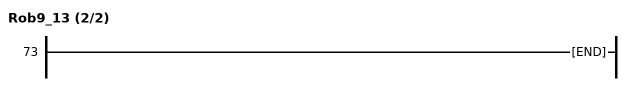
73    END
END_PROGRAM

PROGRAM Rob_12
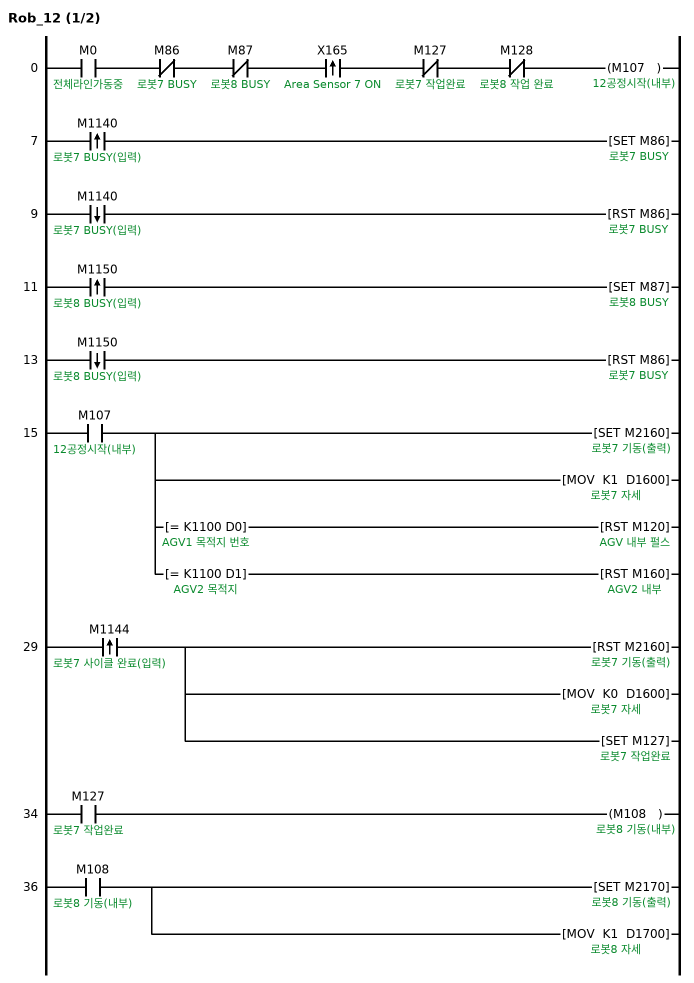
0     LD      M0  ; 전체라인가동중
      ANI     M86  ; 로봇7 BUSY
      ANI     M87  ; 로봇8 BUSY
      ANDP    X165  ; Area Sensor 7 ON
      ANI     M127  ; 로봇7 작업완료
      ANI     M128  ; 로봇8 작업 완료
      OUT     M107  ; 12공정시작(내부)
7     LDP     M1140  ; 로봇7 BUSY(입력)
      SET     M86  ; 로봇7 BUSY
9     LDF     M1140  ; 로봇7 BUSY(입력)
      RST     M86  ; 로봇7 BUSY
11    LDP     M1150  ; 로봇8 BUSY(입력)
      SET     M87  ; 로봇8 BUSY
13    LDF     M1150  ; 로봇8 BUSY(입력)
      RST     M86  ; 로봇7 BUSY
15    LD      M107  ; 12공정시작(내부)
      SET     M2160  ; 로봇7 기동(출력)
      MOV     K1 D1600  ; 로봇7 자세
      MPS
      AND=    K1100 D0  ; AGV1 목적지 번호
      RST     M120  ; AGV 내부 펄스
      MPP
      AND=    K1100 D1  ; AGV2 목적지
      RST     M160  ; AGV2 내부
29    LDP     M1144  ; 로봇7 사이클 완료(입력)
      RST     M2160  ; 로봇7 기동(출력)
      MOV     K0 D1600
      SET     M127  ; 로봇7 작업완료
34    LD      M127  ; 로봇7 작업완료
      OUT     M108  ; 로봇8 기동(내부)
36    LD      M108  ; 로봇8 기동(내부)
      SET     M2170  ; 로봇8 기동(출력)
      MOV     K1 D1700  ; 로봇8 자세
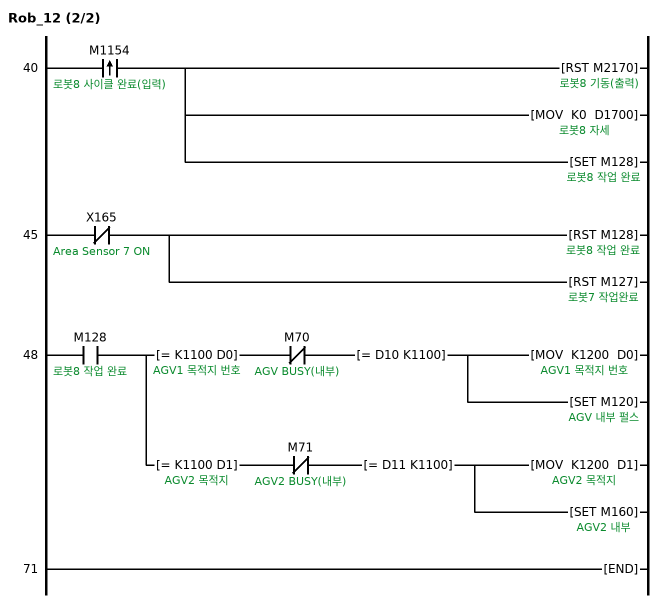
40    LDP     M1154  ; 로봇8 사이클 완료(입력)
      RST     M2170  ; 로봇8 기동(출력)
      MOV     K0 D1700
      SET     M128  ; 로봇8 작업 완료
45    LDI     X165  ; Area Sensor 7 ON
      RST     M128  ; 로봇8 작업 완료
      RST     M127  ; 로봇7 작업완료
48    LD      M128  ; 로봇8 작업 완료
      MPS
      AND=    K1100 D0  ; AGV1 목적지 번호
      ANI     M70  ; AGV BUSY(내부)
      AND=    D10 K1100
      MOV     K1200 D0
      SET     M120  ; AGV 내부 펄스
      MPP
      AND=    K1100 D1  ; AGV2 목적지
      ANI     M71  ; AGV2 BUSY(내부)
      AND=    D11 K1100
      MOV     K1200 D1
      SET     M160  ; AGV2 내부
71    END
END_PROGRAM

// device comments not shown above
X10  ; 로봇4 BUSY
X80  ; 로봇1 BUSY
X84  ; 로봇1 사이클 완료
X8A  ; 로봇2 BUSY
X8E  ; 로봇2 사이클 완료
X93  ; Area Sensor2 ON
X95  ; 로봇3 BUSY
X99  ; 로봇3 사이클 완료
X120  ; 로봇4 BUSY 신호
X124  ; 로봇4 사이클 완료
X129  ; Area Sensor4 ON
X12A  ; 로봇5 BUSY
X12E  ; 로봇5 사이클 완료
X132  ; 로봇6 BUSY
X136  ; 로봇6 사이클 완료
X13C  ; 로봇7 BUSY
X160  ; 로봇7 사이클 완료
X164  ; 로봇8 BUSY
X168  ; 로봇8 사이클 완료
X16C  ; 로봇9 BUSY
X16D  ; 로봇8 사이클 완료
X170  ; 로봇9 사이클 완료
X17B  ; 프레스 Ready
X17D  ; Area Sensor ON
X17E  ; 프레스 사이클 완료
X200  ; AGV BUSY
X201  ; AGV READY
X207  ; 도착완료
Y2  ; ㄹ
Y2D  ; 챔버1 열림
Y2E  ; 챔버2 열림
Y2F  ; 챔버3 열림
Y30  ; 챔버4 열림
Y71  ; 챔버1 닫기
Y72  ; 챔버2 닫기
Y73  ; 챔버3 닫기
Y74  ; 챔버 4 닫기
Y100  ; 로봇1 기동 시작
Y10A  ; 로봇2 기동 시작
Y115  ; 로봇3 기동 시작
Y140  ; 로봇4 기동 시작
Y14A  ; 로봇5 기동 시작
Y155  ; 로봇6 기동 시작
Y180  ; 로봇7 기동 시작
Y18A  ; 로봇8 기동 시작
Y193  ; 로봇9 기동 시작
Y19D  ; 프레스 기동 시작
Y225  ; AGV 기동 시작
M15  ; 경유위치 이동 완료
M100  ; 로봇1 기동 시작
M131  ; 로봇2 작업완료
M170  ; AGV1 명령 수신가능
M171  ; AGV2 명령 수신 가능
M200  ; AGV BUSY
M302  ; 문닫힘신호1
M305  ; 문닫힘 신호2
M308  ; 문닫힘 신호3
M311  ; 문닫힘 신호4
M1110  ; 로봇4 BUSY(입력)
M1139  ; AreaSensor6
M1240  ; 로봇5 기동(출력)
D1300  ; 로봇4 자세
T0  ; 챔버 카운터
T9  ; 수작업7
T10  ; 수작업9
T11  ; 수작업11
T20  ; AGV 딜레이 신호
T41  ; 경유명령 해제
T51  ; 로봇2 대기
